{attribute 'pack_mode' := '1'}
TYPE CETA_Measurement_block2_t :
STRUCT
    Program_number       : USINT;
    Result_chanel_1      : USINT;
    Test_mode            : USINT;
    Result_chanel_2      : USINT;
    Cons_Num_Res_Block   : USINT;
    Num_Following_Blocks : USINT;
    Reserve              : USINT;
    Time_hour            : USINT;
    Time_minute          : USINT;
    Time_second          : USINT;
    Data_offset_12       : CETA_Res_Data_t;
    Data_offset_16       : CETA_Res_Data_t;
    Data_offset_20       : CETA_Res_Data_t;
    Data_offset_24       : CETA_Res_Data_t;
    Data_offset_28       : CETA_Res_Data_t;
    Data_offset_32       : CETA_Res_Data_t;
    Data_offset_36       : CETA_Res_Data_t;
    Data_offset_40       : CETA_Res_Data_t;
    Data_offset_44       : CETA_Res_Data_t;
END_STRUCT
END_TYPE

(* stored: Version 1.1.0.1, ProductVersion 3.1.4024.6
   DUT CETA_Measurement_block2_t: Id {f61c1932-3ecc-41c8-af40-e887d38222d9} *)
